FUNCTION_BLOCK UA_DisconnectWrapper IMPLEMENTS I_OPCUA_Disconnect
VAR_INPUT
END_VAR
VAR_OUTPUT
END_VAR
VAR
	uaDisconnect : UA_Disconnect;
END_VAR

{warning 'add method implementation '}
METHOD start : BOOL
VAR_INPUT
	Execute			: BOOL;
	ConnectionHdl	: DWORD;
	Timeout			: TIME := DEFAULT_ADS_TIMEOUT;
END_VAR
VAR_OUTPUT
	Done	: BOOL;
	Busy	: BOOL;
	Error	: BOOL;
	ErrorID	: DWORD;
END_VAR
uaDisconnect(Execute			:= Execute,
             ConnectionHdl	:= ConnectionHdl,
             Timeout			:= Timeout,
			 Done			=> Done,
			 Busy			=> Busy,
             Error			=> Error,
             ErrorID 		=> ErrorID);
END_METHOD

END_FUNCTION_BLOCK

(* stored: Version 1.1.0.1, ProductVersion 3.1.4024.9
   POU UA_DisconnectWrapper: Id {058e23e6-de7c-42c1-be6f-aae2d049649d}, SpecialFunc None
   Method start: Id {14e71585-8a6f-4ba0-b4b2-3d032087d3a4} *)
